// TIA Portal project "final_code" (V16)

(* hardware
DEVICE "S7-1200 station_1"  S7-1200 Station
   slot 0: "Rack_0"  S7-1200 Rack  Rack  V1.0
   slot 1: "PLC_1"  CPU 1214C DC/DC/DC  6ES7 214-1AG40-0XB0  V4.4
*)

// ===== PLC "PLC_1"  CPU 1214C DC/DC/DC =====

VAR_GLOBAL   // PLC tag table "Default tag table"
   "Tag_1" AT %M200.0 : Bool;
   "Tag_2" AT %M200.1 : Bool;
END_VAR

VAR_GLOBAL   // PLC tag table "input"
   "b_start" AT %I1.5 : Bool;
   "b_stop" AT %I1.4 : Bool;
   "dung" AT %I0.7 : Bool;
   "cb_xylanh_cao" AT %I0.5 : Bool;
   "cb_xylanh_tb" AT %I0.6 : Bool;
   "cb_chieucao" AT %IW64 : Int;
END_VAR

VAR_GLOBAL   // PLC tag table "m_input"
   "m_start" AT %M0.0 : Bool;
   "m_stop" AT %M0.1 : Bool;
   "m_cb_cao" AT %M0.2 : Bool;
   "m_cb_tb" AT %M0.3 : Bool;
   "m_dung" AT %M0.4 : Bool;
   "m_chieucao" AT %MD100 : Real;
   "chieucao_out" AT %MD104 : Real;
   "chieucao_real" AT %MD108 : Real;
   "sosanh" AT %MD112 : Real;
   "so_sp_cao" AT %MW116 : Int;
   "so_sp_thap" AT %MW120 : Int;
   "so_sp_tb" AT %MW124 : Int;
   "m_reset" AT %M0.5 : Bool;
   "gtri_mau" AT %MD128 : Real;
   "m_thap" AT %M0.6 : Bool;
END_VAR

VAR_GLOBAL   // PLC tag table "output"
   "bangtai" AT %Q0.1 : Bool;
   "xylanh_cao" AT %Q1.0 : Bool;
   "xyanh_tb" AT %Q1.1 : Bool;
END_VAR

VAR_GLOBAL   // PLC tag table "m_output"
   "ht_khoidong" AT %M50.0 : Bool;
   "ht_dung" AT %M50.1 : Bool;
   "m_xylanh_cao" AT %M50.2 : Bool;
   "m_xylanh_tb" AT %M50.3 : Bool;
   "m_bangtai" AT %M50.4 : Bool;
END_VAR

DATA_BLOCK "Data_Alarm"   // DB9
{ S7_Optimized_Access := 'FALSE' }
VERSION : 0.1
   VAR
      alarm_1 : Array[0..7] of Bool;
   END_VAR
BEGIN
END_DATA_BLOCK

// folder: System blocks/Program resources

DATA_BLOCK "Timer1"   // DB1
{ S7_Optimized_Access := 'TRUE' }
AUTHOR : Simatic
FAMILY : IEC
NAME : IEC_TMR
VERSION : 1.0
// stored: InstanceOfName IEC_TIMER
"IEC_TIMER"
BEGIN
END_DATA_BLOCK

DATA_BLOCK "Timer2"   // DB2
{ S7_Optimized_Access := 'TRUE' }
AUTHOR : Simatic
FAMILY : IEC
NAME : IEC_TMR
VERSION : 1.0
// stored: InstanceOfName IEC_TIMER
"IEC_TIMER"
BEGIN
END_DATA_BLOCK

DATA_BLOCK "Timer3"   // DB3
{ S7_Optimized_Access := 'TRUE' }
AUTHOR : Simatic
FAMILY : IEC
NAME : IEC_TMR
VERSION : 1.0
// stored: InstanceOfName IEC_TIMER
"IEC_TIMER"
BEGIN
END_DATA_BLOCK

DATA_BLOCK "counter1"   // DB4
{ S7_Optimized_Access := 'TRUE' }
AUTHOR : Simatic
FAMILY : IEC
NAME : CNTR
VERSION : 1.0
// stored: InstanceOfName IEC_COUNTER
"IEC_COUNTER"
BEGIN
END_DATA_BLOCK

DATA_BLOCK "counter2"   // DB5
{ S7_Optimized_Access := 'TRUE' }
AUTHOR : Simatic
FAMILY : IEC
NAME : CNTR
VERSION : 1.0
// stored: InstanceOfName IEC_COUNTER
"IEC_COUNTER"
BEGIN
END_DATA_BLOCK

DATA_BLOCK "counter3"   // DB6
{ S7_Optimized_Access := 'TRUE' }
AUTHOR : Simatic
FAMILY : IEC
NAME : CNTR
VERSION : 1.0
// stored: InstanceOfName IEC_COUNTER
"IEC_COUNTER"
BEGIN
END_DATA_BLOCK

DATA_BLOCK "Timer_cao"   // DB7
{ S7_Optimized_Access := 'TRUE' }
AUTHOR : Simatic
FAMILY : IEC
NAME : IEC_TMR
VERSION : 1.0
// stored: InstanceOfName IEC_TIMER
"IEC_TIMER"
BEGIN
END_DATA_BLOCK

DATA_BLOCK "Timer_tb"   // DB8
{ S7_Optimized_Access := 'TRUE' }
AUTHOR : Simatic
FAMILY : IEC
NAME : IEC_TMR
VERSION : 1.0
// stored: InstanceOfName IEC_TIMER
"IEC_TIMER"
BEGIN
END_DATA_BLOCK

// folder: (top level)

ORGANIZATION_BLOCK "Main"   // OB1, LAD, ProgramCycle
TITLE = "Main Program Sweep (Cycle)"
{ S7_Optimized_Access := 'TRUE' }
VERSION : 0.1
   VAR_INPUT
      Initial_Call : Bool;   // Initial call of this OB
      Remanence : Bool;   // =True, if remanent data are available
   END_VAR
   VAR_TEMP   // added for the SCL form of the ladder/FBD networks
      _w1 : Bool;
   END_VAR
BEGIN

REGION Network 1: khoi dong he thong
   // khoi dong
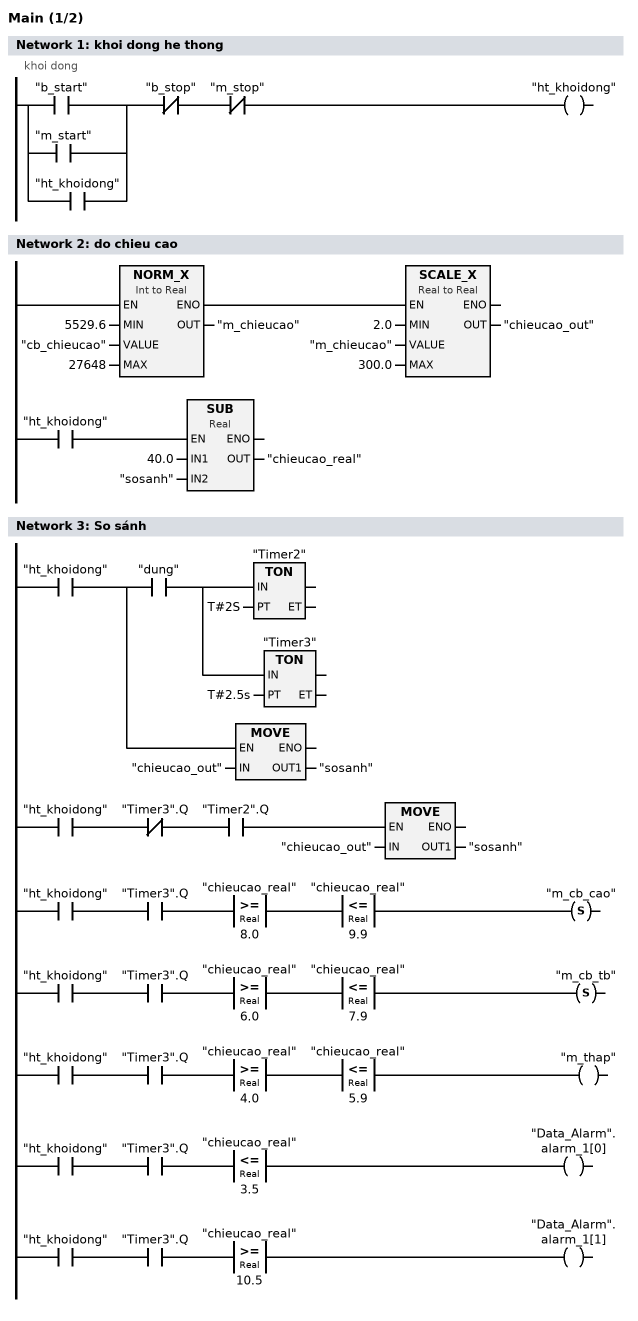
   RUNG wire#powerrail
      Contact( "b_start" )
      wire#w1
      I_Contact( "b_stop" )
      I_Contact( "m_stop" )
      Coil( "ht_khoidong" )
   END_RUNG
   RUNG wire#powerrail
      Contact( "m_start" )
   END_RUNG wire#w1
   RUNG wire#powerrail
      Contact( "ht_khoidong" )
   END_RUNG wire#w1
   // the same network as SCL:
   "ht_khoidong" := ("b_start" OR "m_start" OR "ht_khoidong") AND NOT "b_stop" AND NOT "m_stop";
END_REGION

REGION Network 2: do chieu cao
   RUNG wire#powerrail
      { S7_Templates := "[SrcType := Int, DestType := Real]" } Normalize(min := 5529.6, value := "cb_chieucao", max := 27648, out => "m_chieucao")
      { S7_Templates := "[SrcType := Real, DestType := Real]" } Scale(min := 2.0, value := "m_chieucao", max := 300.0, out => "chieucao_out")
   END_RUNG
   RUNG wire#powerrail
      Contact( "ht_khoidong" )
      { S7_Templates := "SrcType := Real" } Sub(in1 := 40.0, in2 := "sosanh", out => "chieucao_real")
   END_RUNG
   // the same network as SCL:
   "m_chieucao" := NORM_X(MIN := 5529.6, VALUE := "cb_chieucao", MAX := 27648);
   "chieucao_out" := SCALE_X(MIN := 2.0, VALUE := "m_chieucao", MAX := 300.0);
   IF "ht_khoidong" THEN "chieucao_real" := 40.0 - "sosanh"; END_IF;
END_REGION

REGION Network 3: So sánh
   #_w1 := "ht_khoidong" AND "dung";
   "Timer2".TON(IN := #_w1, PT := T#2S);
   "Timer3".TON(IN := #_w1, PT := T#2.5s);
   IF "ht_khoidong" THEN "sosanh" := "chieucao_out"; END_IF;
   IF "ht_khoidong" AND NOT "Timer3".Q AND "Timer2".Q THEN "sosanh" := "chieucao_out"; END_IF;
   IF "ht_khoidong" AND "Timer3".Q AND ("chieucao_real" >= 8.0) AND ("chieucao_real" <= 9.9) THEN
       "m_cb_cao" := TRUE;
   END_IF;
   IF "ht_khoidong" AND "Timer3".Q AND ("chieucao_real" >= 6.0) AND ("chieucao_real" <= 7.9) THEN
       "m_cb_tb" := TRUE;
   END_IF;
   "m_thap" := "ht_khoidong" AND "Timer3".Q AND ("chieucao_real" >= 4.0) AND ("chieucao_real" <= 5.9);
   "Data_Alarm".alarm_1[0] := "ht_khoidong" AND "Timer3".Q AND ("chieucao_real" <= 3.5);
   "Data_Alarm".alarm_1[1] := "ht_khoidong" AND "Timer3".Q AND ("chieucao_real" >= 10.5);
END_REGION

REGION Network 4: dung bang tai
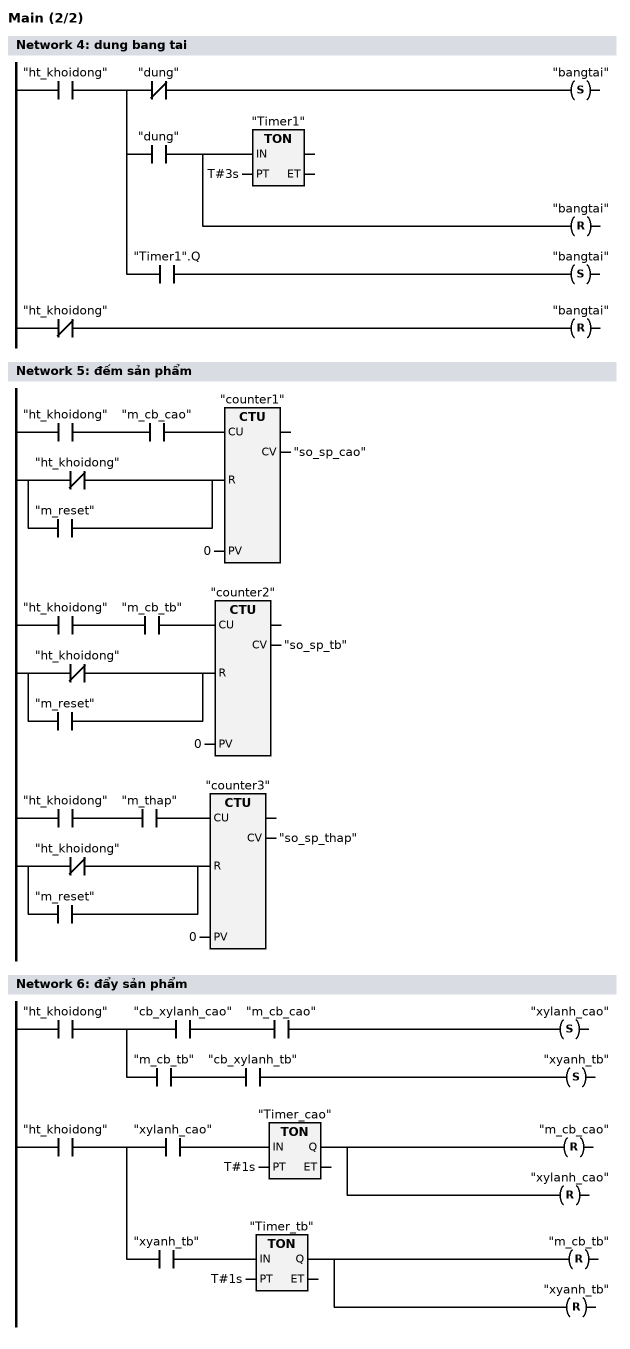
   IF "ht_khoidong" AND NOT "dung" THEN "bangtai" := TRUE; END_IF;
   #_w1 := "ht_khoidong" AND "dung";
   "Timer1".TON(IN := #_w1, PT := T#3s);
   IF #_w1 THEN "bangtai" := FALSE; END_IF;
   IF "ht_khoidong" AND "Timer1".Q THEN "bangtai" := TRUE; END_IF;
   IF NOT "ht_khoidong" THEN "bangtai" := FALSE; END_IF;
END_REGION

REGION Network 5: đếm sản phẩm
   "counter1".CTU(CU := "ht_khoidong" AND "m_cb_cao",
                  R := NOT "ht_khoidong" OR "m_reset",
                  PV := 0,
                  CV => "so_sp_cao");
   "counter2".CTU(CU := "ht_khoidong" AND "m_cb_tb",
                  R := NOT "ht_khoidong" OR "m_reset",
                  PV := 0,
                  CV => "so_sp_tb");
   "counter3".CTU(CU := "ht_khoidong" AND "m_thap",
                  R := NOT "ht_khoidong" OR "m_reset",
                  PV := 0,
                  CV => "so_sp_thap");
END_REGION

REGION Network 6: đẩy sản phẩm
   IF "ht_khoidong" AND "cb_xylanh_cao" AND "m_cb_cao" THEN "xylanh_cao" := TRUE; END_IF;
   IF "ht_khoidong" AND "m_cb_tb" AND "cb_xylanh_tb" THEN "xyanh_tb" := TRUE; END_IF;
   "Timer_cao".TON(IN := "ht_khoidong" AND "xylanh_cao", PT := T#1s);
   IF "Timer_cao".Q THEN
       "m_cb_cao" := FALSE;
       "xylanh_cao" := FALSE;
   END_IF;
   "Timer_tb".TON(IN := "ht_khoidong" AND "xyanh_tb", PT := T#1s);
   IF "Timer_tb".Q THEN
       "m_cb_tb" := FALSE;
       "xyanh_tb" := FALSE;
   END_IF;
END_REGION
END_ORGANIZATION_BLOCK